TYPE ST_ThNTZ_Stellwert :
STRUCT
	Betrieb		: BOOL;
	Leistung	: REAL;
END_STRUCT
END_TYPE

(* stored: Version 1.1.0.1, ProductVersion 3.1.4024.9
   DUT ST_ThNTZ_Stellwert: Id {41cf4a3d-f044-439c-bce9-0bb4eca38016} *)
